// TIA Portal V16 export
// export: Created 2022-12-12T11:14:07.5975361Z, ExportSetting WithDefaults, DisplayName Totally Integrated Automation Portal, DisplayVersion V16 Update 6, DisplayName TIA Portal Version Control Interface, DisplayVersion V16 Update 2, DisplayName TIA Portal Openness, DisplayVersion V16 Update 6, DisplayName SINAMICS Startdrive Advanced, DisplayVersion V16 Update 5, DisplayName SINAMICS Startdrive G130, G150, S120, S150, SINAMICS MV, S210, DisplayVersion V16 Update 5, DisplayName SINAMICS Startdrive G110M, G120, G120C, G120D, G120P, G115D, DisplayVersion V16 Update 5, DisplayName STEP 7 Professional, DisplayVersion V16 Update 6, DisplayName STEP 7 Safety, DisplayVersion V16, DisplayName WinCC Advanced, DisplayVersion V16 Update 6
FUNCTION "FC00_SupportIn" : Void   // FC0, LAD
TITLE = Input support memory
{ S7_Optimized_Access := 'FALSE' }
AUTHOR : Robopac
VERSION : 0.0
// stored: AutoNumber false, IsIECCheckEnabled false, SetENOAutomatically false, UDAEnableTagReadback false
   VAR_TEMP
      AC1 : Int;
      AC2 : Int;
   END_VAR
BEGIN

REGION Network 1: STANDARD
END_REGION

REGION Network 2: Pressure switch (Technoplat)
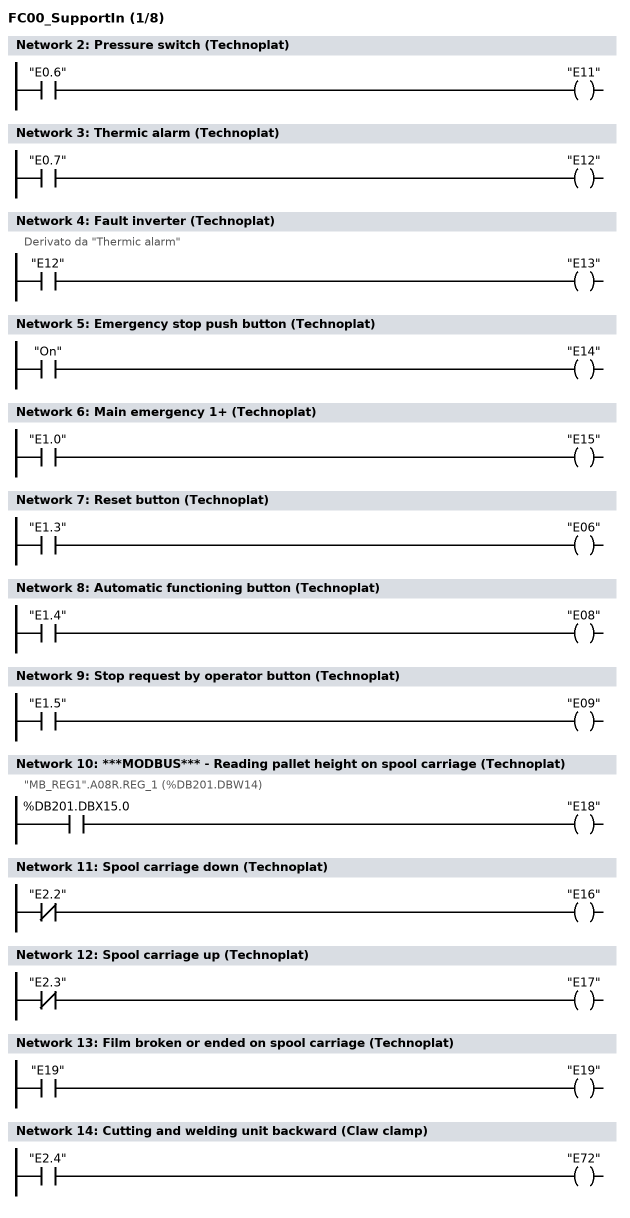
   RUNG wire#powerrail
      Contact( "E0.6" )
      Coil( "E11" )
   END_RUNG
   // the same network as SCL:
   "E11" := "E0.6";
END_REGION

REGION Network 3: Thermic alarm (Technoplat)
   RUNG wire#powerrail
      Contact( "E0.7" )
      Coil( "E12" )
   END_RUNG
   // the same network as SCL:
   "E12" := "E0.7";
END_REGION

REGION Network 4: Fault inverter (Technoplat)
   // Derivato da "Thermic alarm"
   RUNG wire#powerrail
      Contact( "E12" )
      Coil( "E13" )
   END_RUNG
   // the same network as SCL:
   "E13" := "E12";
END_REGION

REGION Network 5: Emergency stop push button (Technoplat)
   RUNG wire#powerrail
      Contact( "On" )
      Coil( "E14" )
   END_RUNG
   // the same network as SCL:
   "E14" := "On";
END_REGION

REGION Network 6: Main emergency 1+ (Technoplat)
   RUNG wire#powerrail
      Contact( "E1.0" )
      Coil( "E15" )
   END_RUNG
   // the same network as SCL:
   "E15" := "E1.0";
END_REGION

REGION Network 7: Reset button (Technoplat)
   RUNG wire#powerrail
      Contact( "E1.3" )
      Coil( "E06" )
   END_RUNG
   // the same network as SCL:
   "E06" := "E1.3";
END_REGION

REGION Network 8: Automatic functioning button (Technoplat)
   RUNG wire#powerrail
      Contact( "E1.4" )
      Coil( "E08" )
   END_RUNG
   // the same network as SCL:
   "E08" := "E1.4";
END_REGION

REGION Network 9: Stop request by operator button (Technoplat)
   RUNG wire#powerrail
      Contact( "E1.5" )
      Coil( "E09" )
   END_RUNG
   // the same network as SCL:
   "E09" := "E1.5";
END_REGION

REGION Network 10: ***MODBUS*** - Reading pallet height on spool carriage (Technoplat)
   // "MB_REG1".A08R.REG_1 (%DB201.DBW14)
   RUNG wire#powerrail
      Contact( %DB201.DBX15.0 )
      Coil( "E18" )
   END_RUNG
   // the same network as SCL:
   "E18" := %DB201.DBX15.0;
END_REGION

REGION Network 11: Spool carriage down (Technoplat)
   RUNG wire#powerrail
      I_Contact( "E2.2" )
      Coil( "E16" )
   END_RUNG
   // the same network as SCL:
   "E16" := NOT "E2.2";
END_REGION

REGION Network 12: Spool carriage up (Technoplat)
   RUNG wire#powerrail
      I_Contact( "E2.3" )
      Coil( "E17" )
   END_RUNG
   // the same network as SCL:
   "E17" := NOT "E2.3";
END_REGION

REGION Network 13: Film broken or ended on spool carriage (Technoplat)
   RUNG wire#powerrail
      Contact( "E19" )
      Coil( "E19" )
   END_RUNG
   // the same network as SCL:
   "E19" := "E19";
END_REGION

REGION Network 14: Cutting and welding unit backward (Claw clamp)
   RUNG wire#powerrail
      Contact( "E2.4" )
      Coil( "E72" )
   END_RUNG
   // the same network as SCL:
   "E72" := "E2.4";
END_REGION

REGION Network 15: Cutting and welding unit forward (Claw clamp)
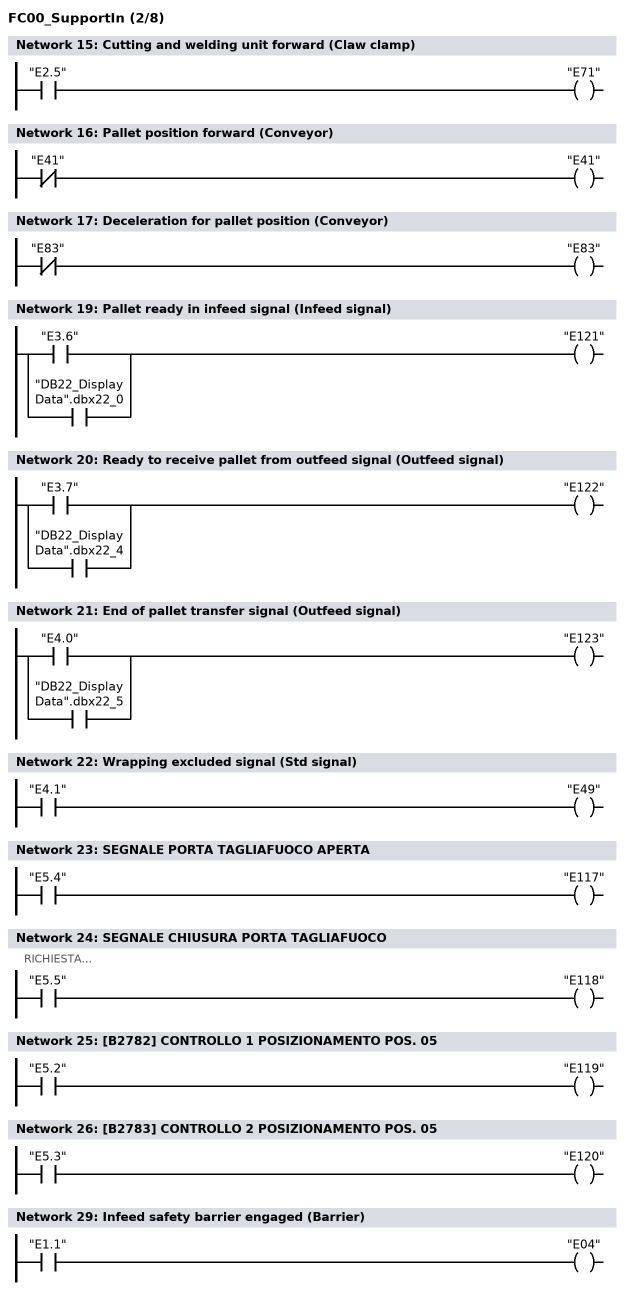
   RUNG wire#powerrail
      Contact( "E2.5" )
      Coil( "E71" )
   END_RUNG
   // the same network as SCL:
   "E71" := "E2.5";
END_REGION

REGION Network 16: Pallet position forward (Conveyor)
   RUNG wire#powerrail
      I_Contact( "E41" )
      Coil( "E41" )
   END_RUNG
   // the same network as SCL:
   "E41" := NOT "E41";
END_REGION

REGION Network 17: Deceleration for pallet position (Conveyor)
   RUNG wire#powerrail
      I_Contact( "E83" )
      Coil( "E83" )
   END_RUNG
   // the same network as SCL:
   "E83" := NOT "E83";
END_REGION

REGION Network 18: EXCHANGE SIGNALS
END_REGION

REGION Network 19: Pallet ready in infeed signal (Infeed signal)
   RUNG wire#powerrail
      Contact( "E3.6" )
      wire#w1
      Coil( "E121" )
   END_RUNG
   RUNG wire#powerrail
      Contact( "DB22_DisplayData".dbx22_0 )
   END_RUNG wire#w1
   // the same network as SCL:
   "E121" := "E3.6" OR "DB22_DisplayData".dbx22_0;
END_REGION

REGION Network 20: Ready to receive pallet from outfeed signal (Outfeed signal)
   RUNG wire#powerrail
      Contact( "E3.7" )
      wire#w1
      Coil( "E122" )
   END_RUNG
   RUNG wire#powerrail
      Contact( "DB22_DisplayData".dbx22_4 )
   END_RUNG wire#w1
   // the same network as SCL:
   "E122" := "E3.7" OR "DB22_DisplayData".dbx22_4;
END_REGION

REGION Network 21: End of pallet transfer signal (Outfeed signal)
   RUNG wire#powerrail
      Contact( "E4.0" )
      wire#w1
      Coil( "E123" )
   END_RUNG
   RUNG wire#powerrail
      Contact( "DB22_DisplayData".dbx22_5 )
   END_RUNG wire#w1
   // the same network as SCL:
   "E123" := "E4.0" OR "DB22_DisplayData".dbx22_5;
END_REGION

REGION Network 22: Wrapping excluded signal (Std signal)
   RUNG wire#powerrail
      Contact( "E4.1" )
      Coil( "E49" )
   END_RUNG
   // the same network as SCL:
   "E49" := "E4.1";
END_REGION

REGION Network 23: SEGNALE PORTA TAGLIAFUOCO APERTA
   RUNG wire#powerrail
      Contact( "E5.4" )
      Coil( "E117" )
   END_RUNG
   // the same network as SCL:
   "E117" := "E5.4";
END_REGION

REGION Network 24: SEGNALE CHIUSURA PORTA TAGLIAFUOCO
   // RICHIESTA...
   RUNG wire#powerrail
      Contact( "E5.5" )
      Coil( "E118" )
   END_RUNG
   // the same network as SCL:
   "E118" := "E5.5";
END_REGION

REGION Network 25: [B2782] CONTROLLO 1 POSIZIONAMENTO POS. 05
   RUNG wire#powerrail
      Contact( "E5.2" )
      Coil( "E119" )
   END_RUNG
   // the same network as SCL:
   "E119" := "E5.2";
END_REGION

REGION Network 26: [B2783] CONTROLLO 2 POSIZIONAMENTO POS. 05
   RUNG wire#powerrail
      Contact( "E5.3" )
      Coil( "E120" )
   END_RUNG
   // the same network as SCL:
   "E120" := "E5.3";
END_REGION

REGION Network 27: ACCESSORIES
END_REGION

REGION Network 28: ***BARRIERS***
END_REGION

REGION Network 29: Infeed safety barrier engaged (Barrier)
   RUNG wire#powerrail
      Contact( "E1.1" )
      Coil( "E04" )
   END_RUNG
   // the same network as SCL:
   "E04" := "E1.1";
END_REGION

REGION Network 30: Outfeed safety barrier engaged (Barrier)
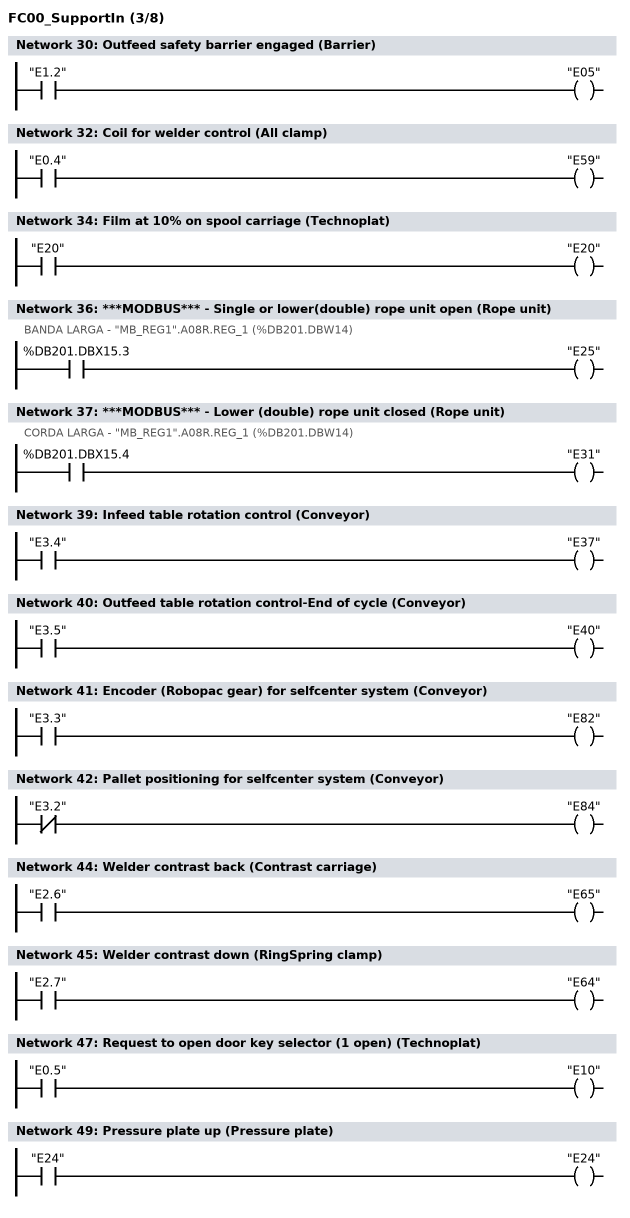
   RUNG wire#powerrail
      Contact( "E1.2" )
      Coil( "E05" )
   END_RUNG
   // the same network as SCL:
   "E05" := "E1.2";
END_REGION

REGION Network 31: ***WELDER***
END_REGION

REGION Network 32: Coil for welder control (All clamp)
   RUNG wire#powerrail
      Contact( "E0.4" )
      Coil( "E59" )
   END_RUNG
   // the same network as SCL:
   "E59" := "E0.4";
END_REGION

REGION Network 33: ***ES_FILM***
END_REGION

REGION Network 34: Film at 10% on spool carriage (Technoplat)
   RUNG wire#powerrail
      Contact( "E20" )
      Coil( "E20" )
   END_RUNG
   // the same network as SCL:
   "E20" := "E20";
END_REGION

REGION Network 35: ***BAND/ROPE***
END_REGION

REGION Network 36: ***MODBUS*** - Single or lower(double) rope unit open (Rope unit)
   // BANDA LARGA - "MB_REG1".A08R.REG_1 (%DB201.DBW14)
   RUNG wire#powerrail
      Contact( %DB201.DBX15.3 )
      Coil( "E25" )
   END_RUNG
   // the same network as SCL:
   "E25" := %DB201.DBX15.3;
END_REGION

REGION Network 37: ***MODBUS*** - Lower (double) rope unit closed (Rope unit)
   // CORDA LARGA - "MB_REG1".A08R.REG_1 (%DB201.DBW14)
   RUNG wire#powerrail
      Contact( %DB201.DBX15.4 )
      Coil( "E31" )
   END_RUNG
   // the same network as SCL:
   "E31" := %DB201.DBX15.4;
END_REGION

REGION Network 38: ***SELF-CENTER***
END_REGION

REGION Network 39: Infeed table rotation control (Conveyor)
   RUNG wire#powerrail
      Contact( "E3.4" )
      Coil( "E37" )
   END_RUNG
   // the same network as SCL:
   "E37" := "E3.4";
END_REGION

REGION Network 40: Outfeed table rotation control-End of cycle (Conveyor)
   RUNG wire#powerrail
      Contact( "E3.5" )
      Coil( "E40" )
   END_RUNG
   // the same network as SCL:
   "E40" := "E3.5";
END_REGION

REGION Network 41: Encoder (Robopac gear) for selfcenter system (Conveyor)
   RUNG wire#powerrail
      Contact( "E3.3" )
      Coil( "E82" )
   END_RUNG
   // the same network as SCL:
   "E82" := "E3.3";
END_REGION

REGION Network 42: Pallet positioning for selfcenter system (Conveyor)
   RUNG wire#powerrail
      I_Contact( "E3.2" )
      Coil( "E84" )
   END_RUNG
   // the same network as SCL:
   "E84" := NOT "E3.2";
END_REGION

REGION Network 43: ***CONTRAST***
END_REGION

REGION Network 44: Welder contrast back (Contrast carriage)
   RUNG wire#powerrail
      Contact( "E2.6" )
      Coil( "E65" )
   END_RUNG
   // the same network as SCL:
   "E65" := "E2.6";
END_REGION

REGION Network 45: Welder contrast down (RingSpring clamp)
   RUNG wire#powerrail
      Contact( "E2.7" )
      Coil( "E64" )
   END_RUNG
   // the same network as SCL:
   "E64" := "E2.7";
END_REGION

REGION Network 46: ***DOOR***
END_REGION

REGION Network 47: Request to open door key selector (1 open) (Technoplat)
   RUNG wire#powerrail
      Contact( "E0.5" )
      Coil( "E10" )
   END_RUNG
   // the same network as SCL:
   "E10" := "E0.5";
END_REGION

REGION Network 48: ***PRESSURE***
END_REGION

REGION Network 49: Pressure plate up (Pressure plate)
   RUNG wire#powerrail
      Contact( "E24" )
      Coil( "E24" )
   END_RUNG
   // the same network as SCL:
   "E24" := "E24";
END_REGION

REGION Network 50: Pressure plate positioning
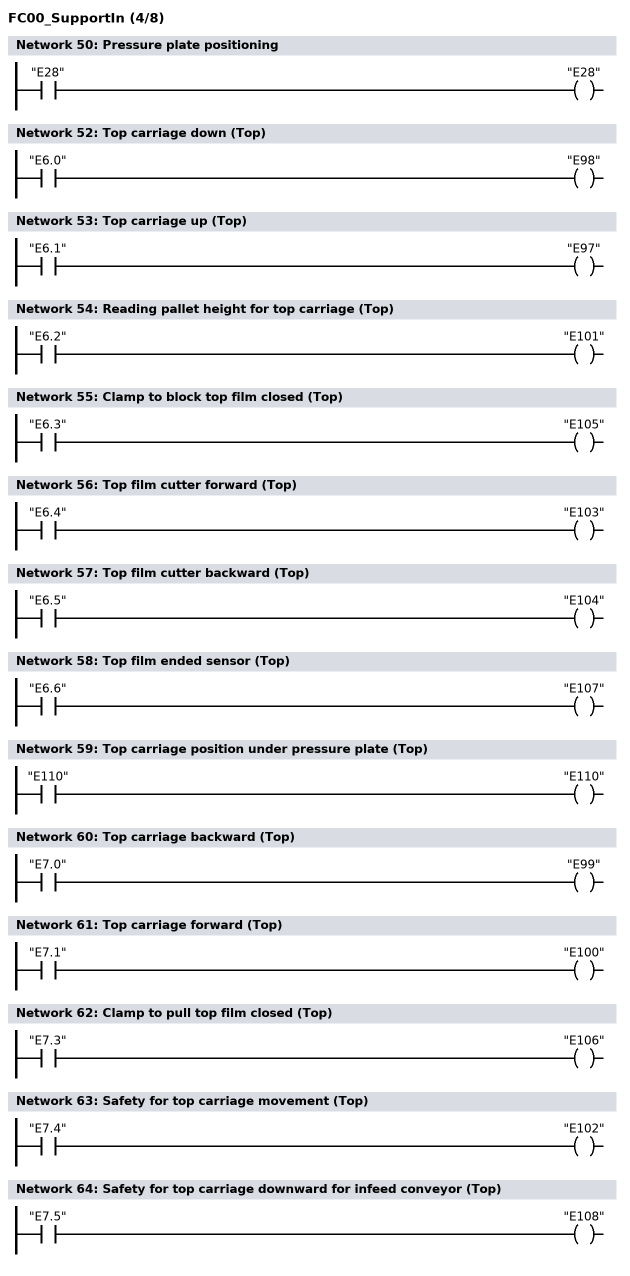
   RUNG wire#powerrail
      Contact( "E28" )
      Coil( "E28" )
   END_RUNG
   // the same network as SCL:
   "E28" := "E28";
END_REGION

REGION Network 51: ***TOP***
END_REGION

REGION Network 52: Top carriage down (Top)
   RUNG wire#powerrail
      Contact( "E6.0" )
      Coil( "E98" )
   END_RUNG
   // the same network as SCL:
   "E98" := "E6.0";
END_REGION

REGION Network 53: Top carriage up (Top)
   RUNG wire#powerrail
      Contact( "E6.1" )
      Coil( "E97" )
   END_RUNG
   // the same network as SCL:
   "E97" := "E6.1";
END_REGION

REGION Network 54: Reading pallet height for top carriage (Top)
   RUNG wire#powerrail
      Contact( "E6.2" )
      Coil( "E101" )
   END_RUNG
   // the same network as SCL:
   "E101" := "E6.2";
END_REGION

REGION Network 55: Clamp to block top film closed (Top)
   RUNG wire#powerrail
      Contact( "E6.3" )
      Coil( "E105" )
   END_RUNG
   // the same network as SCL:
   "E105" := "E6.3";
END_REGION

REGION Network 56: Top film cutter forward (Top)
   RUNG wire#powerrail
      Contact( "E6.4" )
      Coil( "E103" )
   END_RUNG
   // the same network as SCL:
   "E103" := "E6.4";
END_REGION

REGION Network 57: Top film cutter backward (Top)
   RUNG wire#powerrail
      Contact( "E6.5" )
      Coil( "E104" )
   END_RUNG
   // the same network as SCL:
   "E104" := "E6.5";
END_REGION

REGION Network 58: Top film ended sensor (Top)
   RUNG wire#powerrail
      Contact( "E6.6" )
      Coil( "E107" )
   END_RUNG
   // the same network as SCL:
   "E107" := "E6.6";
END_REGION

REGION Network 59: Top carriage position under pressure plate (Top)
   RUNG wire#powerrail
      Contact( "E110" )
      Coil( "E110" )
   END_RUNG
   // the same network as SCL:
   "E110" := "E110";
END_REGION

REGION Network 60: Top carriage backward (Top)
   RUNG wire#powerrail
      Contact( "E7.0" )
      Coil( "E99" )
   END_RUNG
   // the same network as SCL:
   "E99" := "E7.0";
END_REGION

REGION Network 61: Top carriage forward (Top)
   RUNG wire#powerrail
      Contact( "E7.1" )
      Coil( "E100" )
   END_RUNG
   // the same network as SCL:
   "E100" := "E7.1";
END_REGION

REGION Network 62: Clamp to pull top film closed (Top)
   RUNG wire#powerrail
      Contact( "E7.3" )
      Coil( "E106" )
   END_RUNG
   // the same network as SCL:
   "E106" := "E7.3";
END_REGION

REGION Network 63: Safety for top carriage movement (Top)
   RUNG wire#powerrail
      Contact( "E7.4" )
      Coil( "E102" )
   END_RUNG
   // the same network as SCL:
   "E102" := "E7.4";
END_REGION

REGION Network 64: Safety for top carriage downward for infeed conveyor (Top)
   RUNG wire#powerrail
      Contact( "E7.5" )
      Coil( "E108" )
   END_RUNG
   // the same network as SCL:
   "E108" := "E7.5";
END_REGION

REGION Network 65: Safety for top carriage downward for outfeed conveyor (Top)
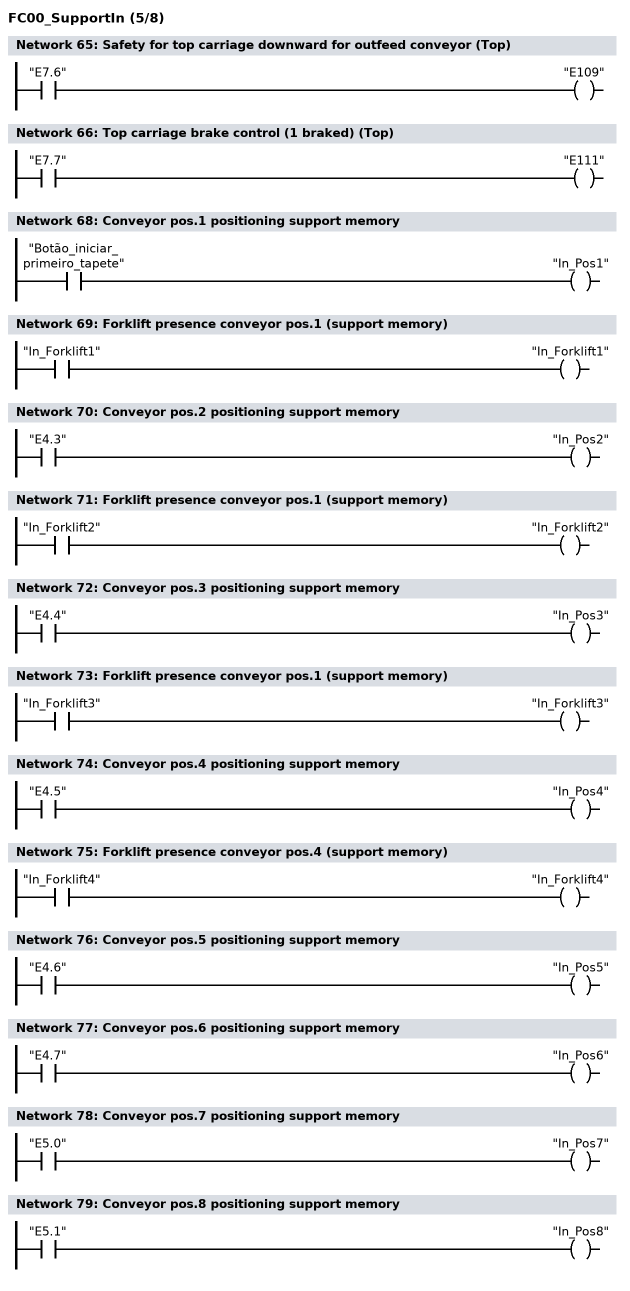
   RUNG wire#powerrail
      Contact( "E7.6" )
      Coil( "E109" )
   END_RUNG
   // the same network as SCL:
   "E109" := "E7.6";
END_REGION

REGION Network 66: Top carriage brake control (1 braked) (Top)
   RUNG wire#powerrail
      Contact( "E7.7" )
      Coil( "E111" )
   END_RUNG
   // the same network as SCL:
   "E111" := "E7.7";
END_REGION

REGION Network 67: ***CONVEYORS***
END_REGION

REGION Network 68: Conveyor pos.1 positioning support memory
   RUNG wire#powerrail
      Contact( "Botão_iniciar_primeiro_tapete" )
      Coil( "In_Pos1" )
   END_RUNG
   // the same network as SCL:
   "In_Pos1" := "Botão_iniciar_primeiro_tapete";
END_REGION

REGION Network 69: Forklift presence conveyor pos.1 (support memory)
   RUNG wire#powerrail
      Contact( "In_Forklift1" )
      Coil( "In_Forklift1" )
   END_RUNG
   // the same network as SCL:
   "In_Forklift1" := "In_Forklift1";
END_REGION

REGION Network 70: Conveyor pos.2 positioning support memory
   RUNG wire#powerrail
      Contact( "E4.3" )
      Coil( "In_Pos2" )
   END_RUNG
   // the same network as SCL:
   "In_Pos2" := "E4.3";
END_REGION

REGION Network 71: Forklift presence conveyor pos.1 (support memory)
   RUNG wire#powerrail
      Contact( "In_Forklift2" )
      Coil( "In_Forklift2" )
   END_RUNG
   // the same network as SCL:
   "In_Forklift2" := "In_Forklift2";
END_REGION

REGION Network 72: Conveyor pos.3 positioning support memory
   RUNG wire#powerrail
      Contact( "E4.4" )
      Coil( "In_Pos3" )
   END_RUNG
   // the same network as SCL:
   "In_Pos3" := "E4.4";
END_REGION

REGION Network 73: Forklift presence conveyor pos.1 (support memory)
   RUNG wire#powerrail
      Contact( "In_Forklift3" )
      Coil( "In_Forklift3" )
   END_RUNG
   // the same network as SCL:
   "In_Forklift3" := "In_Forklift3";
END_REGION

REGION Network 74: Conveyor pos.4 positioning support memory
   RUNG wire#powerrail
      Contact( "E4.5" )
      Coil( "In_Pos4" )
   END_RUNG
   // the same network as SCL:
   "In_Pos4" := "E4.5";
END_REGION

REGION Network 75: Forklift presence conveyor pos.4 (support memory)
   RUNG wire#powerrail
      Contact( "In_Forklift4" )
      Coil( "In_Forklift4" )
   END_RUNG
   // the same network as SCL:
   "In_Forklift4" := "In_Forklift4";
END_REGION

REGION Network 76: Conveyor pos.5 positioning support memory
   RUNG wire#powerrail
      Contact( "E4.6" )
      Coil( "In_Pos5" )
   END_RUNG
   // the same network as SCL:
   "In_Pos5" := "E4.6";
END_REGION

REGION Network 77: Conveyor pos.6 positioning support memory
   RUNG wire#powerrail
      Contact( "E4.7" )
      Coil( "In_Pos6" )
   END_RUNG
   // the same network as SCL:
   "In_Pos6" := "E4.7";
END_REGION

REGION Network 78: Conveyor pos.7 positioning support memory
   RUNG wire#powerrail
      Contact( "E5.0" )
      Coil( "In_Pos7" )
   END_RUNG
   // the same network as SCL:
   "In_Pos7" := "E5.0";
END_REGION

REGION Network 79: Conveyor pos.8 positioning support memory
   RUNG wire#powerrail
      Contact( "E5.1" )
      Coil( "In_Pos8" )
   END_RUNG
   // the same network as SCL:
   "In_Pos8" := "E5.1";
END_REGION

REGION Network 80: OTHER
END_REGION

REGION Network 81: Table rotation phase sensor (Technoplat)
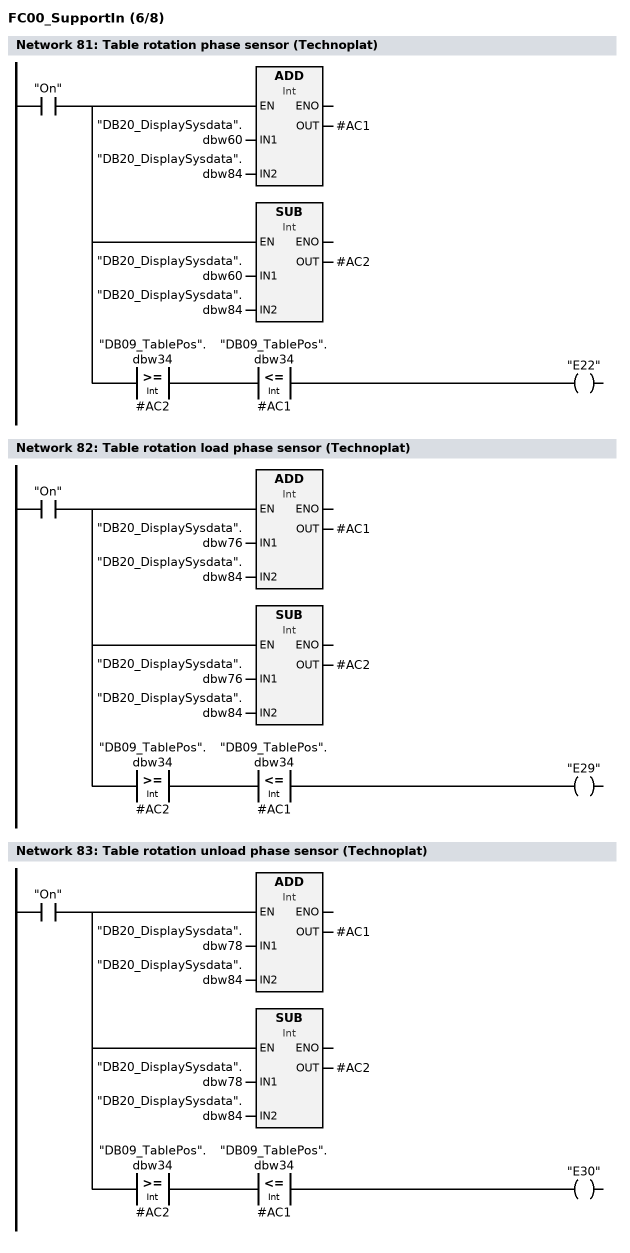
   RUNG wire#powerrail
      Contact( "On" )
      wire#w1
      { S7_Templates := "SrcType := Int"; S7_GenerateENO := "TRUE" } Add(in1 := "DB20_DisplaySysdata".dbw60, in2 := "DB20_DisplaySysdata".dbw84, out => #AC1)
   END_RUNG
   RUNG wire#w1
      { S7_Templates := "SrcType := Int"; S7_GenerateENO := "TRUE" } Sub(in1 := "DB20_DisplaySysdata".dbw60, in2 := "DB20_DisplaySysdata".dbw84, out => #AC2)
   END_RUNG
   RUNG wire#w1
      { S7_Templates := "SrcType := Int" } GE_Contact(in1 := "DB09_TablePos".dbw34, in2 := #AC2)
      { S7_Templates := "SrcType := Int" } LE_Contact(in1 := "DB09_TablePos".dbw34, in2 := #AC1)
      Coil( "E22" )
   END_RUNG
   // the same network as SCL:
   IF "On" THEN
       #AC1 := "DB20_DisplaySysdata".dbw60 + "DB20_DisplaySysdata".dbw84;
       #AC2 := "DB20_DisplaySysdata".dbw60 - "DB20_DisplaySysdata".dbw84;
   END_IF;
   "E22" := "On" AND ("DB09_TablePos".dbw34 >= #AC2) AND ("DB09_TablePos".dbw34 <= #AC1);
END_REGION

REGION Network 82: Table rotation load phase sensor (Technoplat)
   RUNG wire#powerrail
      Contact( "On" )
      wire#w1
      { S7_Templates := "SrcType := Int"; S7_GenerateENO := "TRUE" } Add(in1 := "DB20_DisplaySysdata".dbw76, in2 := "DB20_DisplaySysdata".dbw84, out => #AC1)
   END_RUNG
   RUNG wire#w1
      { S7_Templates := "SrcType := Int"; S7_GenerateENO := "TRUE" } Sub(in1 := "DB20_DisplaySysdata".dbw76, in2 := "DB20_DisplaySysdata".dbw84, out => #AC2)
   END_RUNG
   RUNG wire#w1
      { S7_Templates := "SrcType := Int" } GE_Contact(in1 := "DB09_TablePos".dbw34, in2 := #AC2)
      { S7_Templates := "SrcType := Int" } LE_Contact(in1 := "DB09_TablePos".dbw34, in2 := #AC1)
      Coil( "E29" )
   END_RUNG
   // the same network as SCL:
   IF "On" THEN
       #AC1 := "DB20_DisplaySysdata".dbw76 + "DB20_DisplaySysdata".dbw84;
       #AC2 := "DB20_DisplaySysdata".dbw76 - "DB20_DisplaySysdata".dbw84;
   END_IF;
   "E29" := "On" AND ("DB09_TablePos".dbw34 >= #AC2) AND ("DB09_TablePos".dbw34 <= #AC1);
END_REGION

REGION Network 83: Table rotation unload phase sensor (Technoplat)
   RUNG wire#powerrail
      Contact( "On" )
      wire#w1
      { S7_Templates := "SrcType := Int"; S7_GenerateENO := "TRUE" } Add(in1 := "DB20_DisplaySysdata".dbw78, in2 := "DB20_DisplaySysdata".dbw84, out => #AC1)
   END_RUNG
   RUNG wire#w1
      { S7_Templates := "SrcType := Int"; S7_GenerateENO := "TRUE" } Sub(in1 := "DB20_DisplaySysdata".dbw78, in2 := "DB20_DisplaySysdata".dbw84, out => #AC2)
   END_RUNG
   RUNG wire#w1
      { S7_Templates := "SrcType := Int" } GE_Contact(in1 := "DB09_TablePos".dbw34, in2 := #AC2)
      { S7_Templates := "SrcType := Int" } LE_Contact(in1 := "DB09_TablePos".dbw34, in2 := #AC1)
      Coil( "E30" )
   END_RUNG
   // the same network as SCL:
   IF "On" THEN
       #AC1 := "DB20_DisplaySysdata".dbw78 + "DB20_DisplaySysdata".dbw84;
       #AC2 := "DB20_DisplaySysdata".dbw78 - "DB20_DisplaySysdata".dbw84;
   END_IF;
   "E30" := "On" AND ("DB09_TablePos".dbw34 >= #AC2) AND ("DB09_TablePos".dbw34 <= #AC1);
END_REGION

REGION Network 84: Table rotation phase sensor (Technoplat)
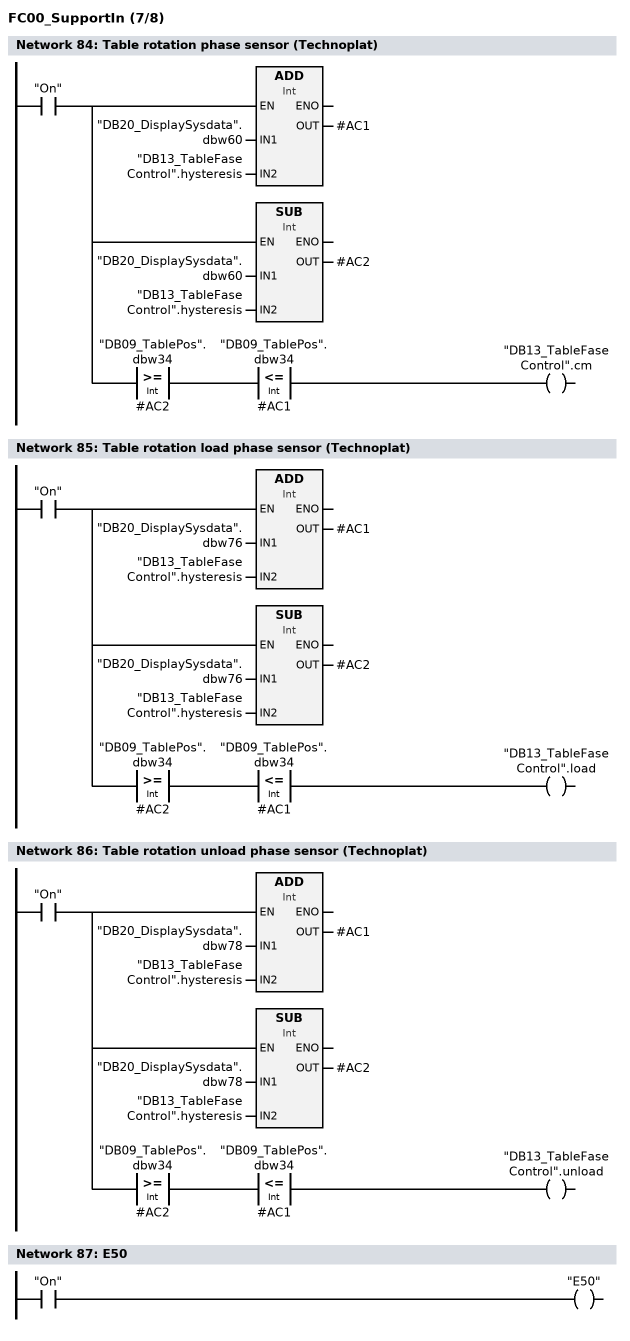
   RUNG wire#powerrail
      Contact( "On" )
      wire#w1
      { S7_Templates := "SrcType := Int"; S7_GenerateENO := "TRUE" } Add(in1 := "DB20_DisplaySysdata".dbw60, in2 := "DB13_TableFaseControl".hysteresis, out => #AC1)
   END_RUNG
   RUNG wire#w1
      { S7_Templates := "SrcType := Int"; S7_GenerateENO := "TRUE" } Sub(in1 := "DB20_DisplaySysdata".dbw60, in2 := "DB13_TableFaseControl".hysteresis, out => #AC2)
   END_RUNG
   RUNG wire#w1
      { S7_Templates := "SrcType := Int" } GE_Contact(in1 := "DB09_TablePos".dbw34, in2 := #AC2)
      { S7_Templates := "SrcType := Int" } LE_Contact(in1 := "DB09_TablePos".dbw34, in2 := #AC1)
      Coil( "DB13_TableFaseControl".cm )
   END_RUNG
   // the same network as SCL:
   IF "On" THEN
       #AC1 := "DB20_DisplaySysdata".dbw60 + "DB13_TableFaseControl".hysteresis;
       #AC2 := "DB20_DisplaySysdata".dbw60 - "DB13_TableFaseControl".hysteresis;
   END_IF;
   "DB13_TableFaseControl".cm := "On" AND ("DB09_TablePos".dbw34 >= #AC2) AND ("DB09_TablePos".dbw34 <= #AC1);
END_REGION

REGION Network 85: Table rotation load phase sensor (Technoplat)
   RUNG wire#powerrail
      Contact( "On" )
      wire#w1
      { S7_Templates := "SrcType := Int"; S7_GenerateENO := "TRUE" } Add(in1 := "DB20_DisplaySysdata".dbw76, in2 := "DB13_TableFaseControl".hysteresis, out => #AC1)
   END_RUNG
   RUNG wire#w1
      { S7_Templates := "SrcType := Int"; S7_GenerateENO := "TRUE" } Sub(in1 := "DB20_DisplaySysdata".dbw76, in2 := "DB13_TableFaseControl".hysteresis, out => #AC2)
   END_RUNG
   RUNG wire#w1
      { S7_Templates := "SrcType := Int" } GE_Contact(in1 := "DB09_TablePos".dbw34, in2 := #AC2)
      { S7_Templates := "SrcType := Int" } LE_Contact(in1 := "DB09_TablePos".dbw34, in2 := #AC1)
      Coil( "DB13_TableFaseControl".load )
   END_RUNG
   // the same network as SCL:
   IF "On" THEN
       #AC1 := "DB20_DisplaySysdata".dbw76 + "DB13_TableFaseControl".hysteresis;
       #AC2 := "DB20_DisplaySysdata".dbw76 - "DB13_TableFaseControl".hysteresis;
   END_IF;
   "DB13_TableFaseControl".load := "On" AND ("DB09_TablePos".dbw34 >= #AC2) AND ("DB09_TablePos".dbw34 <= #AC1);
END_REGION

REGION Network 86: Table rotation unload phase sensor (Technoplat)
   RUNG wire#powerrail
      Contact( "On" )
      wire#w1
      { S7_Templates := "SrcType := Int"; S7_GenerateENO := "TRUE" } Add(in1 := "DB20_DisplaySysdata".dbw78, in2 := "DB13_TableFaseControl".hysteresis, out => #AC1)
   END_RUNG
   RUNG wire#w1
      { S7_Templates := "SrcType := Int"; S7_GenerateENO := "TRUE" } Sub(in1 := "DB20_DisplaySysdata".dbw78, in2 := "DB13_TableFaseControl".hysteresis, out => #AC2)
   END_RUNG
   RUNG wire#w1
      { S7_Templates := "SrcType := Int" } GE_Contact(in1 := "DB09_TablePos".dbw34, in2 := #AC2)
      { S7_Templates := "SrcType := Int" } LE_Contact(in1 := "DB09_TablePos".dbw34, in2 := #AC1)
      Coil( "DB13_TableFaseControl".unload )
   END_RUNG
   // the same network as SCL:
   IF "On" THEN
       #AC1 := "DB20_DisplaySysdata".dbw78 + "DB13_TableFaseControl".hysteresis;
       #AC2 := "DB20_DisplaySysdata".dbw78 - "DB13_TableFaseControl".hysteresis;
   END_IF;
   "DB13_TableFaseControl".unload := "On" AND ("DB09_TablePos".dbw34 >= #AC2) AND ("DB09_TablePos".dbw34 <= #AC1);
END_REGION

REGION Network 87: E50
   RUNG wire#powerrail
      Contact( "On" )
      Coil( "E50" )
   END_RUNG
   // the same network as SCL:
   "E50" := "On";
END_REGION

REGION Network 88: OLD (NOT USED)
END_REGION

REGION Network 89: Key selector automatic (0)/manual (1) mode (Technoplat)
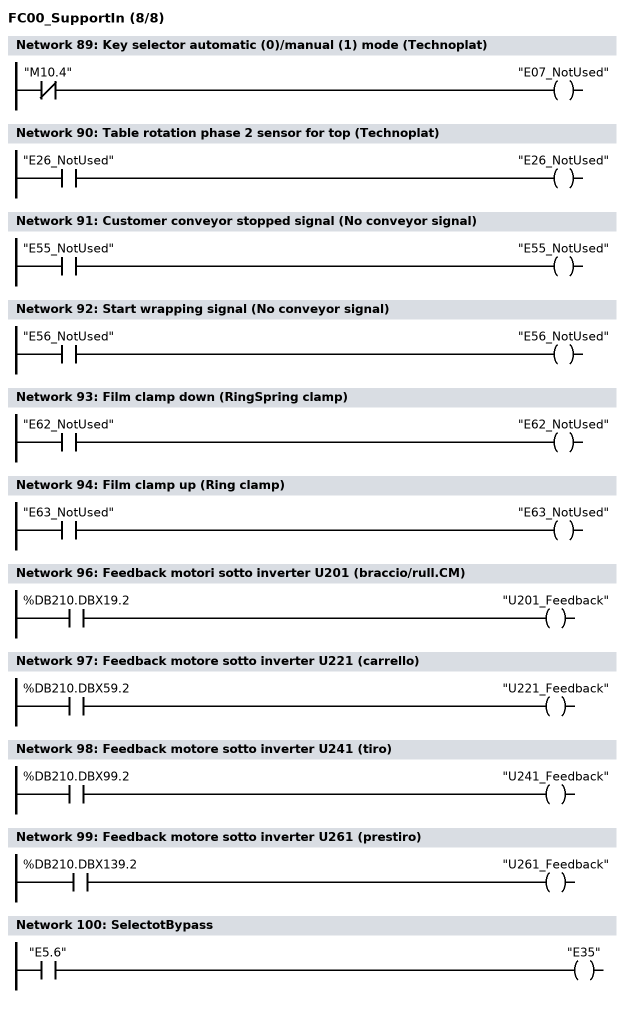
   RUNG wire#powerrail
      I_Contact( "M10.4" )
      Coil( "E07_NotUsed" )
   END_RUNG
   // the same network as SCL:
   "E07_NotUsed" := NOT "M10.4";
END_REGION

REGION Network 90: Table rotation phase 2 sensor for top (Technoplat)
   RUNG wire#powerrail
      Contact( "E26_NotUsed" )
      Coil( "E26_NotUsed" )
   END_RUNG
   // the same network as SCL:
   "E26_NotUsed" := "E26_NotUsed";
END_REGION

REGION Network 91: Customer conveyor stopped signal (No conveyor signal)
   RUNG wire#powerrail
      Contact( "E55_NotUsed" )
      Coil( "E55_NotUsed" )
   END_RUNG
   // the same network as SCL:
   "E55_NotUsed" := "E55_NotUsed";
END_REGION

REGION Network 92: Start wrapping signal (No conveyor signal)
   RUNG wire#powerrail
      Contact( "E56_NotUsed" )
      Coil( "E56_NotUsed" )
   END_RUNG
   // the same network as SCL:
   "E56_NotUsed" := "E56_NotUsed";
END_REGION

REGION Network 93: Film clamp down (RingSpring clamp)
   RUNG wire#powerrail
      Contact( "E62_NotUsed" )
      Coil( "E62_NotUsed" )
   END_RUNG
   // the same network as SCL:
   "E62_NotUsed" := "E62_NotUsed";
END_REGION

REGION Network 94: Film clamp up (Ring clamp)
   RUNG wire#powerrail
      Contact( "E63_NotUsed" )
      Coil( "E63_NotUsed" )
   END_RUNG
   // the same network as SCL:
   "E63_NotUsed" := "E63_NotUsed";
END_REGION

REGION Network 95: PROFINET DATA (inverter)
END_REGION

REGION Network 96: Feedback motori sotto inverter U201 (braccio/rull.CM)
   RUNG wire#powerrail
      Contact( %DB210.DBX19.2 )
      Coil( "U201_Feedback" )
   END_RUNG
   // the same network as SCL:
   "U201_Feedback" := %DB210.DBX19.2;
END_REGION

REGION Network 97: Feedback motore sotto inverter U221 (carrello)
   RUNG wire#powerrail
      Contact( %DB210.DBX59.2 )
      Coil( "U221_Feedback" )
   END_RUNG
   // the same network as SCL:
   "U221_Feedback" := %DB210.DBX59.2;
END_REGION

REGION Network 98: Feedback motore sotto inverter U241 (tiro)
   RUNG wire#powerrail
      Contact( %DB210.DBX99.2 )
      Coil( "U241_Feedback" )
   END_RUNG
   // the same network as SCL:
   "U241_Feedback" := %DB210.DBX99.2;
END_REGION

REGION Network 99: Feedback motore sotto inverter U261 (prestiro)
   RUNG wire#powerrail
      Contact( %DB210.DBX139.2 )
      Coil( "U261_Feedback" )
   END_RUNG
   // the same network as SCL:
   "U261_Feedback" := %DB210.DBX139.2;
END_REGION

REGION Network 100: SelectotBypass
   RUNG wire#powerrail
      Contact( "E5.6" )
      Coil( "E35" )
   END_RUNG
   // the same network as SCL:
   "E35" := "E5.6";
END_REGION
END_FUNCTION
